TYPE ASCF_CC_OPCUACS_Reader_Temp :
STRUCT
	VReal		: ASCF_CC_OPCUACS_Reader_Temp_Real;
	VDInt		: ASCF_CC_OPCUACS_Reader_Temp_Dint;
	VDWord		: ASCF_CC_OPCUACS_Reader_Temp_Dword;
	VBool		: ASCF_CC_OPCUACS_Reader_Temp_Bool;
	VString		: ASCF_CC_OPCUACS_Reader_Temp_String;
END_STRUCT
END_TYPE

(* stored: Version 1.1.0.1, ProductVersion 3.1.4026.4
   DUT ASCF_CC_OPCUACS_Reader_Temp: Id {2a75136e-edf7-4a24-8aac-c0c193fcd9c5} *)
